// TwinCAT 3 PLC project Tub_1
// ProgramVersion: 3.1.4023.0
// libraries:
//   Tc2_ModbusSrv, * (Beckhoff Automation GmbH)
//   Tc2_Standard, * (Beckhoff Automation GmbH)
//   Tc2_System, * (Beckhoff Automation GmbH)
//   Tc2_Utilities, * (Beckhoff Automation GmbH)
//   Tc3_Module, * (Beckhoff Automation GmbH)
// project tree:
//   DUTs/ ST_Alarm.TcDUT, ST_Recipe.TcDUT
//   GVLs/ GVL.TcGVL
//   / PlcTask.TcTTO, RecipeManager.TcRMO (not stored)
//   POUs/ FB_AlarmManager.TcPOU, FB_Furnace.TcPOU, FB_Gantry.TcPOU, FB_Lights.TcPOU, FB_QuenchTank.TcPOU, FB_Recipe.TcPOU, FB_StackLight.TcPOU, FB_Timeout.TcPOU, I_Gantry.TcIO, MAIN.TcPOU
// real-time tasks:
//   TASK PlcTask: cycle T#10ms, priority 20, ADS port 350
// I/O:
//   DEVICE Device 1 (EtherCAT), AmsNetId 5.81.212.44.2.1
//     Term 1 (EK1200) [EK1200-5000 EtherCAT Power supply (2A E-Bus)]
//       Term 2 (EL6070) [EL6070 1Ch. Licensing-Terminal]
//       Term 3 (EL1008) [EL1008 8Ch. Dig. Input 24V, 3ms]
//       Term 4 (EL1008) [EL1008 8Ch. Dig. Input 24V, 3ms]
//       Term 5 (EL2004) [EL2004 4Ch. Dig. Output 24V, 0.5A]
//       Term 6 (EL2008) [EL2008 8Ch. Dig. Output 24V, 0.5A]
//       Term 7 (EL3021) [EL3021 1Ch. Ana. Input 4-20mA DIFF]
//       Term 8 (EL9011) [EL9011 End Terminal]
// variable links:
//   Tub_1/Tub_1 Instance <-> Device 1 (EtherCAT)/Term 1 (EK1200)/Term 5 (EL2004)
//     PlcTask Outputs/GVL.boStackLightGreen <-> Channel 3/Output
//     PlcTask Outputs/GVL.boStackLightRed <-> Channel 1/Output
//     PlcTask Outputs/GVL.boStackLightYellow <-> Channel 2/Output
//   Tub_1/Tub_1 Instance <-> Device 1 (EtherCAT)/Term 1 (EK1200)/Term 7 (EL3021)
//     PlcTask Inputs/GVL.aiSaltTemp <-> AI Standard/Value

CONFIGURATION Tub_1
    RESOURCE PLC ON TwinCAT3
        TASK PlcTask(INTERVAL := T#10ms, PRIORITY := 20);
        PROGRAM MAIN WITH PlcTask : MAIN;
    END_RESOURCE
END_CONFIGURATION

// ---- DUTs/ST_Alarm.TcDUT
TYPE ST_Alarm :
STRUCT
	nAlarmPriority 		: USINT;
	sErrorMsg       	: STRING(50);
	sAlarmID			: STRING(10);
	dtDateAndTime		: DATE_AND_TIME;
END_STRUCT
END_TYPE

// ---- DUTs/ST_Recipe.TcDUT
TYPE ST_Recipe :
STRUCT
	sRecipeName		: STRING(20);
	tHeatSetTime	: TIME;
	tQuenchTime		: TIME;
END_STRUCT
END_TYPE

// ---- GVLs/GVL.TcGVL
{attribute 'qualified_only'}
VAR_GLOBAL

	// general use I/O
	biOperatorDoorClosed 	AT %I* : BOOL;
	biMaintDoorClosed		AT %I* : BOOL;
	
	// stack light I/O
	boStackLightGreen		AT %Q* : BOOL;
	boStackLightYellow		AT %Q* : BOOL;
	boStackLightRed			AT %Q* : BOOL;
	
	// salt furnace I/O
	aiSaltTemp				AT %I* : INT;
	
	// quench tank I/O
	biWaterLevelLow			AT %I* : BOOL;
	biWaterLevelHigh 		AT %I* : BOOL;
	biWaterOverflowAlarm	AT %I* : BOOL;
	biWaterLeakAlarm		AT %I* : BOOL;
	boEnablePump			AT %Q* : BOOL;
	boOpenFillValve			AT %Q* : BOOL;
	boOpenDrainValve		AT %Q* : BOOL;
	boEnableHeaters			AT %Q* : BOOL;
	aiWaterTemp				AT %I* : USINT;
	
	// gantry I/O
	biMotorErrorX			AT %I* : BOOL;
	biMotorErrorY			AT %I* : BOOL;
	
END_VAR

// ---- POUs/I_Gantry.TcIO
INTERFACE I_Gantry

METHOD M_GetPosition : STRING
VAR_INPUT
END_VAR
VAR_OUTPUT
	sCurrentPosition : STRING(20);
END_VAR

(*
	Valid Positions:
	'home' - both axes are at home position by operator door
	'pre heat set' - gantry is above salt bath, waiting to enter
	'setting shape' - tooling fixture is submurged in salt
	'quenching' - tooling fixture is submurged in water
	'moving' - gantry is in motion
	'unknown' - gantry is in unknown position
*)
END_METHOD

METHOD M_GoHeatSet : BOOL
VAR_INPUT
END_VAR
END_METHOD

METHOD M_GoHome : BOOL
VAR_INPUT
END_VAR
END_METHOD

METHOD M_GoPreHeatSet : BOOL
VAR_INPUT
END_VAR
END_METHOD

METHOD M_GoQuench : BOOL
VAR_INPUT
END_VAR
END_METHOD

END_INTERFACE

// ---- POUs/MAIN.TcPOU
PROGRAM MAIN
VAR
	
	// general use variables
	bLocalVar_1				: BOOL;
	bActivateTimeout		: BOOL;
	bHighLevelAlarm			: BOOL;
	bLowLevelAlarm			: BOOL;
	nRetryCounter			: USINT;
	tTotalCycleTime 		: TIME;
	tTimeoutTime			: TIME;
	sMachineState			: STRING(30);
	sPrevMachineState		: STRING(30);
	sErrorMsg				: STRING(50);
	tmrProcessTimer			: Tc2_Standard.TON;
	
	// function block and interface definitions
	fbFurnace 				: FB_Furnace;
	fbGantry 				: FB_Gantry;
	fbQuenchTank 			: FB_QuenchTank;
	fbRecipie				: FB_Recipe;
	fbAlarmManager			: FB_AlarmManager;
	fbTimeout				: FB_Timeout;
	fbStackLight			: FB_StackLight;
	iGantry					: I_Gantry;
	
	// recipe variables
	bCreateRecipe			: BOOL;
	bEditRecipe         	: BOOL;
	bDeleteRecipe			: BOOL;
	tHeatSetTime			: TIME;
	tQuenchTime				: TIME;
	sRecipeName				: STRING(20);
	
	// salt furnace variables
	bSaltCoverOn	    	: BOOL;	
	
	// quench tank variables

END_VAR

// *** GANTRY CONTROL ********************************************************************************

IF sMachineState = 'Startup' THEN
	sMachineState := 'Navigating Home';
	
ELSIF sMachineState = 'Idle' THEN
	sPrevMachineState := 'Idle';

ELSIF sMachineState = 'Navigating to Start Position' THEN
	IF sPrevMachineState <> 'Navigating to Start Position' THEN
		sPrevMachineState := 'Navigating to Start Position';
		iGantry.M_GoPreHeatSet();
		fbTimeout(bActivate := FALSE);
		bActivateTimeout := TRUE;
		tTimeoutTime := T#20S;
		nRetryCounter := 0;
	END_IF

	IF iGantry.M_GetPosition() = 'pre heat set' THEN
		sMachineState := 'Waiting for Start';
	ELSIF fbTimeout.nAttempts >= 3 THEN
		sMachineState := 'Help Required';
		sErrorMsg := 'Unable to move to start pos from home';
	ELSIF fbTimeout.nAttempts > nRetryCounter THEN
		iGantry.M_GoPreHeatSet();
		nRetryCounter := nRetryCounter + 1;
	END_IF

ELSIF sMachineState = 'Waiting for Start' THEN
    RETURN;
	
ELSIF sMachineState = 'Getting Salty' THEN
	IF sPrevMachineState <> 'Getting Salty' THEN
		sPrevMachineState := 'Getting Salty';
	    iGantry.M_GoHeatSet();
		fbTimeout(bActivate := FALSE);
		bActivateTimeout := TRUE;
		tTimeoutTime := T#10S;
		nRetryCounter := 0;
	END_IF

	IF iGantry.M_GetPosition() = 'setting shape' THEN
		sMachineState := 'Heat Soaking';
	ELSIF fbTimeout.nAttempts >= 3 THEN
		sMachineState := 'Help Required';
		sErrorMsg := 'Unable to enter salt bath';
	ELSIF fbTimeout.nAttempts > nRetryCounter THEN
		iGantry.M_GoHeatSet();
		nRetryCounter := nRetryCounter + 1;
	END_IF
	
ELSIF sMachineState = 'Heat Soaking' THEN
	IF sPrevMachineState <> 'Heat Soaking' THEN
		sPrevMachineState := 'Heat Soaking';
		tmrProcessTimer(IN := FALSE);
	END_IF
	
	tmrProcessTimer(IN := TRUE, PT := tHeatSetTime);
	IF tmrProcessTimer.Q THEN
		sMachineState := 'Navigating to Quench';
	END_IF
	
ELSIF sMachineState = 'Navigating to Quench' THEN
	IF sPrevMachineState <> 'Navigating to Quench' THEN
		sPrevMachineState := 'Navigating to Quench';
		iGantry.M_GoQuench();
		fbTimeout(bActivate := FALSE);
		bActivateTimeout := TRUE;
		tTimeoutTime := T#10S;
		nRetryCounter := 0;
	END_IF

	IF iGantry.M_GetPosition() = 'quenching' THEN
		sMachineState := 'Quenching';
	ELSIF fbTimeout.nAttempts >= 3 THEN
		sMachineState := 'Help Required';
		sErrorMsg := 'Unable to navigate from heat to quench';
	ELSIF fbTimeout.nAttempts > nRetryCounter THEN
		iGantry.M_GoHeatSet();
		nRetryCounter := nRetryCounter + 1;
	END_IF	

ELSIF sMachineState = 'Quenching' THEN
	IF sPrevMachineState <> 'Quenching' THEN
		sPrevMachineState := 'Quenching';
		tmrProcessTimer(IN := FALSE);
	END_IF
	
	tmrProcessTimer(IN := TRUE, PT := tQuenchTime);
	IF tmrProcessTimer.Q THEN
		sMachineState := 'Navigating Home';
	END_IF
	
ELSIF sMachineState = 'Navigating Home' THEN
	IF sPrevMachineState <> 'Navigating Home' THEN
		sPrevMachineState := 'Navigating Home';
		iGantry.M_GoHome();
		fbTimeout(bActivate := FALSE);
		bActivateTimeout := TRUE;
		tTimeoutTime := T#20S;
		nRetryCounter := 0;
	END_IF
	
	IF iGantry.M_GetPosition() = 'Home' THEN
		sMachineState := 'Idle';
	ELSIF fbTimeout.nAttempts >= 3 THEN
		sMachineState := 'Help Required';
		sErrorMsg := 'Unable to move to start pos from home';
	ELSIF fbTimeout.nAttempts > nRetryCounter THEN
		iGantry.M_GoPreHeatSet();
		nRetryCounter := nRetryCounter + 1;
	END_IF
	
END_IF

fbTimeout(bActivate := bActivateTimeout, tDuration := tTimeoutTime);


// *** RECIPE ACTIONS *********************************************************************************

IF bCreateRecipe THEN
	bCreateRecipe := FALSE;
	fbRecipie.M_Create(sName := sRecipeName, 
					   tIngredient_1 := tHeatSetTime, 
					   tIngredient_2 := tQuenchTime);
END_IF

IF bEditRecipe THEN
	bEditRecipe := FALSE;
	fbRecipie.M_Edit(sName := sRecipeName, 
					 tNewIngredient_1 := tHeatSetTime, 
					 tNewIngredient_2 := tQuenchTime);
END_IF

IF bDeleteRecipe THEN
	bDeleteRecipe := FALSE;
	fbRecipie.M_Delete(sName := sRecipeName);
END_IF


// *** QUENCH TANK OPERATION ***************************************************************************




// *** STACK LIGHT OPERATION ***************************************************************************

IF sMachineState = 'Idle' THEN
	IF bHighLevelAlarm THEN
		fbStackLight(bBlinkEnabled := FALSE, sColor := 'red');
	ELSIF bLowLevelAlarm THEN
		fbStackLight(bBlinkEnabled := FALSE, sColor := 'yellow');
	ELSE
		fbStackLight(bBlinkEnabled := FALSE, sColor := 'green');
	END_IF	
ELSE
	IF bHighLevelAlarm THEN
		fbStackLight(bBlinkEnabled := TRUE, sColor := 'red');
	ELSIF bLowLevelAlarm THEN
		fbStackLight(bBlinkEnabled := TRUE, sColor := 'yellow');
	ELSE
		fbStackLight(bBlinkEnabled := TRUE, sColor := 'green');
	END_IF	
END_IF

END_PROGRAM

// ---- POUs/FB_Furnace.TcPOU
FUNCTION_BLOCK FB_Furnace
VAR_INPUT
END_VAR
VAR_OUTPUT
END_VAR

END_FUNCTION_BLOCK

// ---- POUs/FB_Gantry.TcPOU
FUNCTION_BLOCK FB_Gantry IMPLEMENTS I_Gantry
VAR_INPUT
	bExecuteHeatSetCycle 	: BOOL;
	bGoHome 				: BOOL;		// nStateVariable 0
	bGoPreHeatSet 			: BOOL;		// nStateVariable 1
	bGoHeatSet 				: BOOL;		// nStateVariable 2
	bGoPreQuench 			: BOOL;		// nStateVariable 3
	bGoQuench 				: BOOL;		// nStateVariable 4
	bStayIdle				: BOOL; 	// nStateVariable 5
END_VAR
VAR_OUTPUT
	bAtHome 				: BOOL;
	bAtPreHeatSet 			: BOOL;
	bAtHeatSet 				: BOOL;
	bAtPreQuench 			: BOOL;
	bAtQuench 				: BOOL;
	bBusy					: BOOL;
	bHeatSetCycleFinished	: BOOL;
END_VAR
VAR
END_VAR

METHOD M_GetPosition : STRING
VAR_INPUT
END_VAR
VAR_OUTPUT
	sCurrentPosition : STRING(20);
END_VAR
END_METHOD

METHOD M_GoHeatSet : BOOL
VAR_INPUT
END_VAR
END_METHOD

METHOD M_GoHome : BOOL
VAR_INPUT
END_VAR
END_METHOD

METHOD M_GoPreHeatSet : BOOL
VAR_INPUT
END_VAR
END_METHOD

METHOD M_GoQuench : BOOL
VAR_INPUT
END_VAR
END_METHOD

END_FUNCTION_BLOCK

// ---- POUs/FB_QuenchTank.TcPOU
FUNCTION_BLOCK FB_QuenchTank
VAR_INPUT
	sAction 				: STRING(10);			// 'fill', 'drain'
END_VAR

VAR_OUTPUT
	bError					: BOOL;
	nWaterTemp				: USINT;				// scaled value of thermocouple
	sErrorMsg				: STRING(60);
END_VAR

VAR
	tDrainTimeout           : TIME := T#10S;		// time until drain is aborted
	tFillTimeout			: TIME := T#10S;		// time until fill is aborted
	tPumpEnableDelay		: TIME := T#3S;			// delay to allow drain valve to open before pump is enabled
	tmrFillTimer			: Tc2_Standard.TON;
	tmrDrainTimer			: Tc2_Standard.TON;
END_VAR

IF sAction = 'fill' THEN
	tmrFillTimer(IN := TRUE, PT := tFillTimeout);
	IF NOT tmrFillTimer.Q THEN
		GVL.boOpenFillValve := TRUE;
		bError := FALSE;
		sErrorMsg := '';
	ELSE
		GVL.boOpenFillValve := FALSE;
		bError := TRUE;
		sErrorMsg := 'Timeout while filling tank - check float high level sensor';
	END_IF

ELSIF sAction = 'drain' THEN
	tmrDrainTimer(IN := TRUE, PT := tDrainTimeout);
	GVL.boOpenDrainValve := TRUE;
	IF tmrDrainTimer.ET > tPumpEnableDelay THEN
		GVL.boEnablePump := TRUE;
	END_IF
ELSE
	tmrDrainTimer(IN := FALSE);
	tmrFillTimer(IN := FALSE);
END_IF

METHOD M_DrainTank : BOOL
VAR_INPUT
END_VAR
END_METHOD

METHOD M_FillTank : BOOL
VAR_INPUT
END_VAR
END_METHOD

END_FUNCTION_BLOCK

// ---- POUs/FB_Recipe.TcPOU
FUNCTION_BLOCK PUBLIC FB_Recipe
VAR_INPUT
	bCreateRecipe		: BOOL;
	bEditRecipe         : BOOL;
	bDeleteRecipe		: BOOL;
	tHeatSetTime		: TIME;
	tQuenchTime			: TIME;
	sRecipeName			: STRING(20);
	stRecipeIn			: ST_Recipe;
END_VAR

VAR_OUTPUT
	stRecipeOut			: ST_Recipe;
END_VAR

VAR
	nCounter_1			: INT;
	nMaxRecipes			: INT := 100;
END_VAR

VAR PERSISTENT 
    aRecipeBook			: ARRAY[1..100] OF ST_Recipe;
	aRecipeNames		: ARRAY[1..100] OF STRING(20);
END_VAR

METHOD M_Create : ST_Recipe
VAR_INPUT
	sName				: STRING(20);
	tIngredient_1 		: TIME;
	tIngredient_2 		: TIME;
	
END_VAR
VAR_OUTPUT
	bCreateSuceessful	:BOOL;
	sErrorMsg			:STRING(30) := 'None';
END_VAR
VAR
	stRecipe			: ST_Recipe;
	nCounter			: INT;
	bDuplicateFound		: BOOL;
END_VAR
// check for duplicates
WHILE NOT (bDuplicateFound) AND (nCounter <= nMaxRecipes) DO
	FOR nCounter := 1 TO nMaxRecipes DO
		IF aRecipeBook[nCounter].sRecipeName = sName THEN
			bDuplicateFound := TRUE;
			sErrorMsg := 'Duplicate recipe name found';
			bCreateSuceessful := FALSE;
		END_IF
	END_FOR
END_WHILE

// check recipe array for empty spot
IF NOT bDuplicateFound THEN
	nCounter := 1;
	WHILE (aRecipeBook[nCounter].sRecipeName <> '') AND (nCounter <= nMaxRecipes) DO
		nCounter := nCounter + 1;
	END_WHILE
	
	// check for full recipe array
	IF nCounter > nMaxRecipes THEN
		sErrorMsg := 'Recipe book full';
		bCreateSuceessful := FALSE;
		
	// if no duplicates, fill next available recipe slot	
	ELSIF NOT bDuplicateFound THEN
		stRecipe.sRecipeName := sName;
		stRecipe.tHeatSetTime := tIngredient_1;
		stRecipe.tQuenchTime := tIngredient_2;
		aRecipeBook[nCounter] := stRecipe;
		bCreateSuceessful := TRUE;
		M_UpdateRecipeNames();
	END_IF
END_IF
END_METHOD

METHOD M_Delete : BOOL
VAR_INPUT
	sName				: STRING(20);
END_VAR
VAR_OUTPUT
	bDeleteSuccessful 	: BOOL;
END_VAR
VAR
	nCounter 			: INT;
END_VAR
nCounter := 1;
WHILE (aRecipeBook[nCounter].sRecipeName <> sName) AND (nCounter <= nMaxRecipes) DO
	nCounter := nCounter + 1;
END_WHILE

IF nCounter > nMaxRecipes THEN
	bDeleteSuccessful := FALSE;
ELSE
	aRecipeBook[nCounter].sRecipeName := '';
	aRecipeBook[nCounter].tHeatSetTime := T#0S;
	aRecipeBook[nCounter].tQuenchTime := T#0S;
	bDeleteSuccessful := TRUE;
	M_UpdateRecipeNames();
END_IF
END_METHOD

METHOD M_Edit : BOOL
VAR_INPUT
	sName				: STRING(20);
	tNewIngredient_1 	: TIME;
	tNewIngredient_2 	: TIME;
END_VAR
VAR_OUTPUT
	bEditSuccessful 	: BOOL;
	sErrorMsg			: STRING(30);
	stRecipeOut			: ST_Recipe;
END_VAR
VAR
	nCounter			: INT := 1;
END_VAR
// find recipe in recipe book
WHILE (aRecipeBook[nCounter].sRecipeName <> sName) AND (nCounter <= nMaxRecipes) DO
	nCounter := nCounter + 1;
END_WHILE

// check if recipe not found
IF nCounter > nMaxRecipes THEN
	sErrorMsg := 'Recipe not found';
	bEditSuccessful := FALSE;
	
// update time values
ELSE
	aRecipeBook[nCounter].tHeatSetTime := tNewIngredient_1;
	aRecipeBook[nCounter].tQuenchTime := tNewIngredient_2;
END_IF
END_METHOD

METHOD M_OrderList : BOOL
VAR_INPUT
	sName			: STRING(20);
END_VAR
VAR
	nCounter		: INT := 1;
	nStrLen_1		: INT;
	nStrLen_2		: INT;
	sString_1		: STRING(20);
	sString_2		: STRING(20);
	sPlaceholder	: STRING(20);
END_VAR
WHILE nCounter < nMaxRecipes DO
	// store nth and nth + 1 string as uppercase
	sString_1 := aRecipeNames[nCounter];
	sString_2 := aRecipeNames[nCounter + 1];
	sString_1 := F_ToUCase(sString_1);
	sString_2 := F_ToUCase(sString_2);
	
	// store string lengths
	nStrLen_1 := LEN(STR := sString_1);
	nStrLen_2 := LEN(STR := sString_2);
	
	// check if 1st string empty and 2nd string not
	IF nStrLen_1 = 0 AND nStrLen_2 <> 0 THEN
		// replcae 1st str with 2nd str
		aRecipeNames[nCounter] := sString_2;
	
	// check if both values are 0
	ELSIF nStrLen_1 = 0 AND nStrLen_2 = 0 THEN
		EXIT;
		
	// check if 1st string 1st char is less than 2nd string 1st char
	ELSIF LEFT(STR := sString_1, SIZE := 1) < LEFT(STR := sString_2, SIZE := 1) THEN 
		// swap names
		sPlaceholder := sString_1;
		aRecipeNames[nCounter] := sString_2;
		aRecipeNames[nCounter + 1] := sPlaceholder;
		nCounter := 1;
	END_IF
	nCounter := nCounter + 1;
END_WHILE
END_METHOD

METHOD M_UpdateRecipeNames : BOOL
VAR_INPUT
END_VAR
VAR
	nItem	: INT;
	nIndex	: INT := 1;
END_VAR
FOR nItem := 1 TO nMaxRecipes DO
	IF aRecipeBook[nItem].sRecipeName <> '' THEN
		aRecipeNames[nIndex] := aRecipeBook[nItem].sRecipeName;
		nIndex := nIndex + 1;
	END_IF
END_FOR
END_METHOD

END_FUNCTION_BLOCK

// ---- POUs/FB_AlarmManager.TcPOU
FUNCTION_BLOCK FB_AlarmManager
VAR_INPUT
END_VAR
VAR_OUTPUT
	aAlarmBuffer			: ARRAY[1..25] OF ST_Alarm;
END_VAR
VAR PERSISTENT
	aAlarmHistory			: ARRAY[1..100] OF ST_Alarm;
END_VAR
VAR
	nAlarmBufferSize		: USINT := 25;
	nAlarmHistorySize 		: USINT := 100;
END_VAR

METHOD M_Add : BOOL
VAR_INPUT
	nAlarmPriority		: USINT;
	sErrorMsg 			: STRING(50);
END_VAR
VAR
	nItem				: USINT;
	nIndex				: USINT := 1;
	stNewAlarm			: ST_Alarm;
	stTempAlarm_1		: ST_Alarm;
	stTempAlarm_2		: ST_Alarm;
END_VAR
// store new alarm into ST_Alarm format
stNewAlarm.nAlarmPriority := nAlarmPriority;
stNewAlarm.sErrorMsg := sErrorMsg;
// stNewAlarm.dtDateAndTime := Tc2_Utilities.SYSTEMTIME_TO_DT;

// store new alarm at top of buffer
stTempAlarm_1 := aAlarmBuffer[1];
aAlarmBuffer[1] := stNewAlarm;
nIndex := 2;

// move all older alarms down
WHILE ((aAlarmBuffer[nItem].sErrorMsg <> '') AND (nIndex < 25)) DO
	stTempAlarm_2 := aAlarmBuffer[nIndex];
	aAlarmBuffer[nIndex] := stTempAlarm_1;
	stTempAlarm_1 := stTempAlarm_2;
	nIndex := nIndex + 1;
END_WHILE
END_METHOD

METHOD M_Dismiss : BOOL
VAR_INPUT
END_VAR
END_METHOD

END_FUNCTION_BLOCK

// ---- POUs/FB_Timeout.TcPOU
FUNCTION_BLOCK FB_Timeout
VAR_INPUT
	bActivate			: BOOL;
	tDuration			: TIME;
END_VAR
VAR_OUTPUT
	nAttempts			: USINT := 0;
END_VAR
VAR
	bTimerEnable		: BOOL := TRUE;
	tmrTimeoutTimer		: Tc2_Standard.TON;
END_VAR

IF bActivate THEN
	tmrTimeoutTimer(IN := bTimerEnable, PT := tDuration);
	IF tmrTimeoutTimer.Q THEN
		nAttempts := nAttempts + 1;
		tmrTimeoutTimer(IN := FALSE);
	END_IF
	
ELSE
	nAttempts := 0;
	bTimerEnable := TRUE;
END_IF

END_FUNCTION_BLOCK

// ---- POUs/FB_StackLight.TcPOU
FUNCTION_BLOCK FB_StackLight
VAR_INPUT
	bBlinkEnabled		: BOOL;
	sColor				: STRING(10);
END_VAR
VAR
	bLightOnCycle		: BOOL;
	tBlinkDelay			: TIME := T#500MS;
	tmrBlinkTimer		: Tc2_Standard.TON;
END_VAR

IF bBlinkEnabled THEN
	tmrBlinkTimer(IN := TRUE, PT := tBlinkDelay);
	IF tmrBlinkTimer.Q AND bLightOnCycle THEN
		bLightOnCycle := FALSE;
		tmrBlinkTimer(IN := FALSE);
		IF sColor = 'red' THEN
			GVL.boStackLightRed := TRUE;
			GVL.boStackLightYellow := FALSE;
			GVL.boStackLightGreen := FALSE;
		ELSIF sColor = 'yellow' THEN
			GVL.boStackLightRed := FALSE;
			GVL.boStackLightYellow := TRUE;
			GVL.boStackLightGreen := FALSE;
		ELSE
			GVL.boStackLightRed := FALSE;
			GVL.boStackLightYellow := FALSE;
			GVL.boStackLightGreen := TRUE;
		END_IF
	ELSIF tmrBlinkTimer.Q AND (NOT bLightOnCycle) THEN
		bLightOnCycle := TRUE;
		tmrBlinkTimer(IN := FALSE);
		GVL.boStackLightRed := FALSE;
		GVL.boStackLightYellow := FALSE;
		GVL.boStackLightGreen := FALSE;
	END_IF
ELSE
	IF sColor = 'red' THEN
		GVL.boStackLightRed := TRUE;
		GVL.boStackLightYellow := FALSE;
		GVL.boStackLightGreen := FALSE;
	ELSIF sColor = 'yellow' THEN
		GVL.boStackLightRed := FALSE;
		GVL.boStackLightYellow := TRUE;
		GVL.boStackLightGreen := FALSE;
	ELSE
		GVL.boStackLightRed := FALSE;
		GVL.boStackLightYellow := FALSE;
		GVL.boStackLightGreen := TRUE;
	END_IF
END_IF

END_FUNCTION_BLOCK

// ---- POUs/FB_Lights.TcPOU
FUNCTION_BLOCK FB_Lights
VAR_INPUT
END_VAR
VAR_OUTPUT
END_VAR
VAR
END_VAR

END_FUNCTION_BLOCK
